// TIA Portal V20 export
// export: Created 2025-12-01T14:57:08.0285312Z, ExportSetting None, DisplayName Totally Integrated Automation Portal, DisplayVersion V20 Update 3, DisplayName TIA Portal Openness, DisplayVersion V20 Update 3, DisplayName TIA Portal Version Control Interface, DisplayVersion V20 Update 3, DisplayName STEP 7 Professional, DisplayVersion V20 Update 3, DisplayName STEP 7 Safety, DisplayVersion V20 Update 2, DisplayName WinCC Basic/Comfort/Advanced, DisplayVersion V20 Update 3, DisplayName WinCC Professional, DisplayVersion V20 Update 3, DisplayName WinCC Unified, DisplayVersion V20 Update 3
FUNCTION "FC980_CTRL_VAR_DANFOSS_PN" : Void   // FC980, STL
TITLE = Comunicación con variador Danfoss Profinet
{ S7_Optimized_Access := 'FALSE' }
AUTHOR : VARIADOR
NAME : 20150506
VERSION : 3.2
// stored: AutoNumber false
   VAR_INPUT
      Numero_Dispositivo : Int;   // numero dispositivo profinet
      Dir_INI : Int;   // Dirección inicio periferia
      DB_Diag_profinet : Int;
      DB_Danfoss : Int;   // DB_CTRL_Danfoss_PN
      Avance : Bool;
      Retroceso : Bool;
      Rearme : Bool;
      Conexion_Estrella : Bool;
      Sentido_Giro : Bool;
      Motor_2 : Bool;
      Salida_Digital : Bool;
      Consigna_Vel : Int;   // 0..327,67hz; 5000 = 50.00Hz
   END_VAR
   VAR_TEMP
      Danfoss_STW : Struct
         Speed_Ok : Bool;
         Bus_Control : Bool;
         Frecuenc_Limit_Ok : Bool;
         In_Operation : Bool;
         N_Drive_Ok : Bool;
         Voltage_Exceeded : Bool;
         Torque_Exceeded : Bool;
         Timer_Exceeded : Bool;
         Control_Ready : Bool;
         Drive_Ready : Bool;
         Enable : Bool;
         Trip : Bool;
         ON_2 : Bool;
         ON_3 : Bool;
         Start_Not_Possible : Bool;
         Warnning : Bool;
      END_STRUCT;
      Danfoss_CTW : Struct
         Jog1 : Bool;
         Jog2 : Bool;
         DataValid : Bool;
         SlowDown : Bool;
         CatchUp : Bool;
         N_ParameterSetUP : Bool;
         N_ParameterSet_UP1 : Bool;
         Reverse : Bool;
         ON1 : Bool;
         ON2 : Bool;
         ON3 : Bool;
         NoCoasting : Bool;
         Ramp : Bool;
         UseRamp : Bool;
         Start : Bool;
         Reset : Bool;
      END_STRUCT;
      Actual_Speed : Int;
      Digital_Input : Word;
      ACC : Int;
      DCC : Int;
      Dig_Output : Struct
         Output_T42 : Bool;
         Reseva_25 : Bool;
         Reserva_26 : Bool;
         Reserva_27 : Bool;
         Reserva_28 : Bool;
         Reserva_29 : Bool;
         Reserva_30 : Bool;
         Reserva_31 : Bool;
         Reserva_32 : Bool;
         Reserva_16 : Bool;
         Reserva_17 : Bool;
         Reserva_18 : Bool;
         Reserva_19 : Bool;
         Reserva_20 : Bool;
         Reserva_21 : Bool;
         Reserva_22 : Bool;
      END_STRUCT;
      Red_Nodo : Struct
         Had_Failed : Bool;
         Deactivadted : Bool;
         Reserved_10 : Bool;
         Reseved_11 : Bool;
         Reserved_12 : Bool;
         Reserved_13 : Bool;
         Reserved_14 : Bool;
         Reserved_15 : Bool;
         OK : Bool;
         Maintenance : Bool;
         Faulty : Bool;
         Failed : Bool;
         Was_Deativated : Bool;
         DPV1 : Bool;
         Was_Under_Maintenace : Bool;
         Was_Failed : Bool;
      END_STRUCT;
      Temp_Consigna_Velocidad : Int;
      Real_Consign_Vel : Real;
      DINT_Consinga_Vel : DInt;
      NDB_Nodos : Word;
      NDB_Variador : Word;
      P_DanfossSTW : DWord;
      Temporal_dint : DInt;
      P_DanfossCTW : DWord;
      P_DigitalOutput : DWord;
      P_RedNodo : DWord;
   END_VAR
BEGIN

NETWORK
TITLE = Inicializar la temporales.
//=======================================================================================================================
// -- Inicializar las variables temporales

      L     P##Danfoss_STW;
      T     #P_DanfossSTW;
      L     P##Danfoss_CTW;
      T     #P_DanfossCTW;
      L     P##Dig_Output;
      T     #P_DigitalOutput;
      L     P##Red_Nodo;
      T     #P_RedNodo;

      L     0;
      T     LW [#P_DanfossSTW];
      T     LW [#P_DanfossCTW];
      T     LW [#P_DigitalOutput];
      T     #Temp_Consigna_Velocidad;
      T     #Actual_Speed;
      T     #Digital_Input;
      L     #DB_Diag_profinet;
      T     #NDB_Nodos;
      L     #DB_Danfoss;
      T     #NDB_Variador;

//=======================================================================================================================

NETWORK
TITLE = Chequeo de activación del simulador
//=======================================================================================================================
// -- Vamos a comprobar si tenemos que ir por la ejecución normal o por la del simulador
      SET;
      AN    "Activar_Simulador";
      JC    NORE;  // ejecución normal de lectura de entradas
//=======================================================================================================================

NETWORK
TITLE = Ejecución SIMULADOR de la lectura de E/S
//=======================================================================================================================
// -- En este segmeto leemos toda la inforamcion del SIMULADOR y lo guardamos en el DB correspondiente

// Calculo puntero datos donde vamos a ir recogiendo la información
      L     #Dir_INI;
      SLD   3;  //Dar formato de Integer a Puntero
      LAR1;


//=======================================================================================================================
// leemos todos los datos de periferia

// Status word
      L     IW [AR1, P#0.0];
      T     LW [#P_DanfossSTW];  // Status word 1

// Velocidad actual
      L     IW [AR1, P#2.0];
      T     #Actual_Speed;

// Entradas Digitales

      L     IW [AR1, P#4.0];
      T     #Digital_Input;  // las señales de las E/S se lean y se dejen dentro de imagen

/////////////////////// Modificacion Pablo 21-04-2017----
//ahora sobreescribiremos, los bits ON2 y ON3, para utilizarlos
//como ON2-> Variador_Activo
//como ON3-> Variador velocidad diferente de 0
      AN    #Danfoss_STW.Start_Not_Possible;
      AN    #Danfoss_STW.Trip;
      A     #Danfoss_STW.Enable;
      =     #Danfoss_STW.ON_2;

      L     #Actual_Speed;
      L     0;
      <>I;
      =     #Danfoss_STW.ON_3;

//=======================================================================================================================
// guardamos los datos en el DB del variador, pero antes calculamos el puntero

      OPN   DB [#NDB_Variador];
      L     #Numero_Dispositivo;
      L     10;  //longitud registro datos
      *I;
      SLD   3;  //3 para pasar a formato puntero
      LAR1;

// guardamos los datos en el DB del variador

      L     LW [#P_DanfossSTW];  //Miramos la posicion del variador y la guardamos en el DB y posicion adecuada.
      T     DBW [AR1, P#0.0];
      L     #Actual_Speed;  //Miramos la posicion del elevador y la guardamos en el DB y posicion adecuada.
      T     DBW [AR1, P#2.0];
      L     #Digital_Input;  //Miramos la posicion del elevador y la guardamos en el DB y posicion adecuada.
      T     DBW [AR1, P#4.0];

//=======================================================================================================================
      JU    CONT;  // saltamos al control del variador
//=======================================================================================================================

NETWORK
TITLE = verificación de nodo presente: Ejecución NORMAL
//=======================================================================================================================
// -- antes de proceder a la lectura del variador diagnosticamos el nodo

NORE: OPN   DB [#NDB_Nodos];
      L     #Numero_Dispositivo;
      L     1;  //longitud registro datos
      -I;
      L     2;  // Longitud de estructura de la DB.
      *I;
      SLD   3;  //3 para pasar a formato puntero
      LAR1;
      L     DBW [AR1, P#0.0];
      T     LW [#P_RedNodo];  // dentro de la zona temporal el w14 tiene el formato del diagnóstico de profinet

      A     #Red_Nodo.OK;
      JC    nxt;  // saltamos al final porque no vamos a leer un variador que no está presente

////////////////////////////////////////////////////////////////////
//Ini Nieves modificado el 26/01/2018
// pasamos a cero todos los datos del variador

      OPN   DB [#NDB_Variador];
      L     #Numero_Dispositivo;
      L     10;  //longitud registro datos
      *I;
      SLD   3;  //3 para pasar a formato puntero
      LAR1;

// guardamos los datos en el DB del variador

      L     0;
      T     DBW [AR1, P#0.0];
      T     DBW [AR1, P#2.0];
      T     DBW [AR1, P#4.0];

      JU    FIN;

// Fin Nieves modificado el 26/01/2018
//=======================================================================================================================

NETWORK
TITLE = Ejecución NORMAL de la lectura de E/S
// En este segmeto leemos toda la inforamcion del Variador y lo guardamos en el DB 
// correspondiente
//=======================================================================================================================
// -- En este segmeto leemos toda la inforamcion del Variador y lo guardamos en el DB correspondiente

// Calculo puntero datos donde vamos a ir recogiendo la información
nxt:  L     #Dir_INI;
      SLD   3;  //Dar formato de Integer a Puntero
      LAR1;


//=======================================================================================================================
// leemos todos los datos de periferia

// Status word
      L     IW [AR1, P#0.0];
      T     LW [#P_DanfossSTW];  // Status word 1

// Velocidad actual
      L     IW [AR1, P#2.0];
      T     #Actual_Speed;

/////////////////////// Modificacion Pablo 21-04-2017----
//ahora sobreescribiremos, los bits ON2 y ON3, para utilizarlos
//como ON2-> Variador_Activo
//como ON3-> Variador velocidad diferente de 0
      A     #Danfoss_STW.Enable;
      A     #Danfoss_STW.Control_Ready;
      A     #Danfoss_STW.Drive_Ready;
      A     #Danfoss_STW.Bus_Control;
      AN    #Danfoss_STW.Trip;
      AN    #Danfoss_STW.Start_Not_Possible;
      =     #Danfoss_STW.ON_2;

      L     #Actual_Speed;
      L     0;
      <>I;
      =     #Danfoss_STW.ON_3;

// Entradas Digitales

      L     IW [AR1, P#4.0];
      T     IW [AR1, P#4.0];  //Nieves: modificación el 01/09/16  estando configurados los variadores fuera de la imagen de proceso,
      T     #Digital_Input;  // las señales de las E/S se lean y se dejen dentro de imagen

//=======================================================================================================================
// Nieves: modificación 02/03/17


      L     ID [AR1, P#8.0];  // dato del los detectores conectados en forma de encoder
      ABS;  // le aplicamos el valor absoluto para eliminar el bit de mayor peso que corresponde al signo
      T     #Temporal_dint;
      T     ID [AR1, P#8.0];  // una vez eliminado el signo lo paso a la zona de imagen de proceso para usarlo

// fin modificación 02/03/17
//=======================================================================================================================
// guardamos los datos en el DB del variador, pero antes calculamos el puntero

      OPN   DB [#NDB_Variador];
      L     #Numero_Dispositivo;
      L     10;  //longitud registro datos
      *I;
      SLD   3;  //3 para pasar a formato puntero
      LAR1;

// guardamos los datos en el DB del variador

      L     LW [#P_DanfossSTW];  //Miramos la posicion del variador y la guardamos en el DB y posicion adecuada.
      T     DBW [AR1, P#0.0];
      L     #Actual_Speed;  //Miramos la posicion del elevador y la guardamos en el DB y posicion adecuada.
      T     DBW [AR1, P#2.0];
      L     #Digital_Input;  //Miramos la posicion del elevador y la guardamos en el DB y posicion adecuada.
      T     DBW [AR1, P#4.0];

//=======================================================================================================================

NETWORK
TITLE = Control del variador
// Control del variador
//=======================================================================================================================
//-- Control del variador

CONT: A     #Danfoss_STW.Control_Ready;
      =     #Danfoss_CTW.ON1;

      SET;
      =     #Danfoss_CTW.ON2;
      =     #Danfoss_CTW.ON3;
      =     #Danfoss_CTW.NoCoasting;
      =     #Danfoss_CTW.Ramp;
      =     #Danfoss_CTW.UseRamp;
      =     #Danfoss_CTW.DataValid;


      CLR;
      =     #Danfoss_CTW.Jog1;
      =     #Danfoss_CTW.Jog2;
      =     #Danfoss_CTW.SlowDown;
      =     #Danfoss_CTW.CatchUp;

//=======================================================================================================================

NETWORK
TITLE = Selección de parametros
// Danfoss tiene la opcion de poder controlar 4 tipos de variadores distintos. 
// Para 
// proteger cada uno de ellos utilizamos la logica entre 2 bits.
// Parameter list 1 y 2 se van a utilizar para el control de 2 motores en triangulo
// Parameter list 3 y 4 se van a utilizar para el control de 2 motores en 
// estrella.
//=======================================================================================================================

//  Danfoss tiene la opcion de poder controlar 4 tipos de variadores distintos.
//  Para proteger cada uno de ellos utilizamos la logica entre 2 bits.
//  Parameter list 1 y 2 se van a utilizar para el control de 2 motores en triangulo
//  Parameter list 3 y 4 se van a utilizar para el control de 2 motores en estrella.

//=======================================================================================================================
// Seleccionar lista de parametros 1

      AN    #Conexion_Estrella;
      AN    #Motor_2;
      JCN   M2;
      R     #Danfoss_CTW.N_ParameterSetUP;
      R     #Danfoss_CTW.N_ParameterSet_UP1;
      JU    MF;

//=======================================================================================================================
// Seleccionar lista de parametros 2

M2:   AN    #Conexion_Estrella;
      A     #Motor_2;
      JCN   M3;
      S     #Danfoss_CTW.N_ParameterSetUP;
      R     #Danfoss_CTW.N_ParameterSet_UP1;
      JU    MF;

//=======================================================================================================================
// Seleccionar lista de parametros 3

M3:   A     #Conexion_Estrella;
      AN    #Motor_2;
      JCN   M4;
      R     #Danfoss_CTW.N_ParameterSetUP;
      S     #Danfoss_CTW.N_ParameterSet_UP1;
      JU    MF;

//=======================================================================================================================
// Seleccionar lista de parametros 4

M4:   A     #Conexion_Estrella;
      A     #Motor_2;
      JCN   MF;
      S     #Danfoss_CTW.N_ParameterSetUP;
      S     #Danfoss_CTW.N_ParameterSet_UP1;


//=======================================================================================================================
MF:   NOP   0;
//=======================================================================================================================


NETWORK
TITLE = Rearme
//=======================================================================================================================
// -- Enviar el rearme al variador

      A     #Rearme;
      =     #Danfoss_CTW.Reset;

//=======================================================================================================================

NETWORK
TITLE = Salida Digital T42
//=======================================================================================================================
// -- Enviar la salida digital

      A     #Salida_Digital;
      =     #Dig_Output.Output_T42;
//=======================================================================================================================


NETWORK
TITLE = El starta se activa tanto en el avance como en el retroceso.
//=======================================================================================================================
// -- El start se activa tanto en el avance como en el retroceso.

      A(;
      O     #Avance;
      O     #Retroceso;
      );
      A     #Danfoss_STW.Control_Ready;
      A     #Danfoss_STW.Control_Ready;
      AN    #Danfoss_STW.Start_Not_Possible;
//    UN    #Danfoss_STW.Warnning
      =     #Danfoss_CTW.Start;

//=======================================================================================================================

NETWORK
TITLE = adaptación del avance y retroceso
// Para que todos los variadores tengan el mismo programa generamos un patilla de 
// sentido de giro para cambiar el sentido desde el PLC y mantener las entradas de 
// Avance y Retroceso
//=======================================================================================================================
// Para que todos los variadores tengan el mismo programa generamos un patilla de
// sentido de giro para cambiar el sentido desde el PLC y mantener las entradas de
// Avance y Retroceso
//=======================================================================================================================
      A     #Sentido_Giro;
      JC    SG;
      A     #Retroceso;
      A     #Danfoss_STW.Control_Ready;
      A     #Danfoss_STW.Control_Ready;
      AN    #Danfoss_STW.Start_Not_Possible;
//    UN    #Danfoss_STW.Warnning
      =     #Danfoss_CTW.Reverse;
      JU    SF;


//=======================================================================================================================
SG:   A     #Avance;
      A     #Danfoss_STW.Control_Ready;
      A     #Danfoss_STW.Control_Ready;
      AN    #Danfoss_STW.Start_Not_Possible;
//      UN    #Danfoss_STW.Warnning
      =     #Danfoss_CTW.Reverse;

//=======================================================================================================================

SF:   NOP   0;

//=======================================================================================================================

NETWORK
TITLE = adaptación de la consigna
// Danfoss funciona en % es para que valla a la velocidad nominal que le hemos 
// puesto en el variador hay que enviarle 16384 por eso hacemos la regla de tres.
// El valor 384 es para un motor en Estrella y sale de la division entre 16384/5000
// 
// El valir 188 es para un motor en Triangulo y sale de la division entre 
// 16384/8700
//=======================================================================================================================
//    Danfoss funciona en % es para que vaya a la velocidad nominal que le hemos
// puesto en el variador hay que enviarle 16384 por eso hacemos la regla de tres.
// El valor 384 es para un motor en Estrella y sale de la division entre 16384/5000(HZ)

//El valor 188 es para un motor en Triangulo y sale de la division entre   16384/8700(HZ)
//=======================================================================================================================


// Convertimos el Entero en doble entero
      L     #Consigna_Vel;
      ITD;
      T     #DINT_Consinga_Vel;

// Convertimos el doble entero en Real
      L     #DINT_Consinga_Vel;
      DTR;
      T     #Real_Consign_Vel;

//Hacemos los calculos en Reales

      A     #Conexion_Estrella;
      JCN   TRI;

      L     #Real_Consign_Vel;
      L     2.34;  //  L     3.2768
      *R;
      T     #Real_Consign_Vel;

      JU    VF;


//=======================================================================================================================
TRI:  L     #Real_Consign_Vel;
      L     1.6382;  //L     1.883
      *R;
      T     #Real_Consign_Vel;

//=======================================================================================================================

// El valor obtenido lo pasamos a Entero

VF:   L     #Real_Consign_Vel;
      RND;
      T     #Temp_Consigna_Velocidad;
//=======================================================================================================================

NETWORK
TITLE = 
//=======================================================================================================================
//-- calculamos el puntero a los datos del variador dentro del DB para recoger los datos antes de escribirlos.

      OPN   DB [#NDB_Variador];
      L     #Numero_Dispositivo;
      L     10;  //longitud registro datos
      *I;
      SLD   3;  //3 para pasar a formato puntero
      LAR1;  // calculamos el puntero a la dirección inicial del variador

// -- ACC Leemos el valor de la Aceleración de la DB

      L     DBW [AR1, P#6.0];  //Miramos la posicion del elevador y la guardamos en el DB y posicion adecuada.
      T     #ACC;

// -- DCC Leemos el valor de la Decelaración de la DB

      L     DBW [AR1, P#8.0];  //Miramos la posicion del elevador y la guardamos en el DB y posicion adecuada.
      T     #DCC;

//=======================================================================================================================
// Calculo puntero datos a la periferia
      L     #Dir_INI;
      SLD   3;  //Dar formato de Integer a Puntero
      LAR1;


//=======================================================================================================================
// -- Vamos a comprobar si tenemos que ir por la ejecución normal o por la del simulador
      SET;
      AN    "Activar_Simulador";
      JC    NORS;
//=======================================================================================================================



NETWORK
TITLE = Ejecución SIMULADOR para la escritura de las salidas
//=======================================================================================================================
// Control Word word
      L     LW [#P_DanfossCTW];
      T     QW [AR1, P#0.0];  // Control Word

// Salida Digital Terminal 42
      L     LW [#P_DigitalOutput];
      T     QW [AR1, P#8.0];  // Salida digital

//=======================================================================================================================
      SET;
      O     #Avance;
      O     #Retroceso;
      JCN   FIN;

// Consigna de velocidad
      L     #Temp_Consigna_Velocidad;
      T     QW [AR1, P#2.0];  // Consigna Velocidad
// ACC
      L     #ACC;
      T     QW [AR1, P#4.0];  // Aceleracion
// DCC
      L     #DCC;
      T     QW [AR1, P#6.0];  // Deceleracion


//=======================================================================================================================
      JU    FIN;

//=======================================================================================================================

NETWORK
TITLE = Ejecución NORMAL para la escritura de las salidas
//=======================================================================================================================
// Control Word word
NORS: L     LW [#P_DanfossCTW];
      T     QW [AR1, P#0.0];  // Control Word

// Salida Digital Terminal 42
      L     LW [#P_DigitalOutput];
      T     QW [AR1, P#8.0];  // Deceleracion

//=======================================================================================================================
      SET;
      O     #Avance;
      O     #Retroceso;
      JCN   FIN;

// Consigna de velocidad
      L     #Temp_Consigna_Velocidad;
      T     QW [AR1, P#2.0];  // Consigna Velocidad
// ACC
      L     #ACC;
      T     QW [AR1, P#4.0];  // Aceleracion
// DCC
      L     #DCC;
      T     QW [AR1, P#6.0];  // Deceleracion

//=======================================================================================================================

NETWORK
TITLE = FIN
//=======================================================================================================================
FIN:  NOP   0;

//=======================================================================================================================


END_FUNCTION
